FUNCTION_BLOCK Handling_Teach EXTENDS TcoCore.TcoSequencer
VAR
	_o : TcoCore.TcoSequencerObserver(THIS^);	
	_dialog : TcoCore.TcoDialog(THIS^);
END_VAR

PROPERTY Components : REFERENCE TO Handling_Components
GET
VAR
    _parent : POINTER TO Handling;
END_VAR
IF __QUERYPOINTER(_ParentObject,_parent) THEN // Check if _Parent is Station001
	Components REF= _parent^._components;              // If the check is successful dereference a pointer. simlar to THIS^ or SUPER^
END_IF
END_GET
END_PROPERTY

(*~
	<docu>
		<summary>
			Main method of the sequener. Custom code needs to be placed here. The sequencer is executed by call of InstanceName.Run() method.
			This method is abstract, and it must be overridden in derived block.
		</summary>
	</docu>
~*)
METHOD PROTECTED  Main : BOOL
VAR
	test: TcEventEntry;
	answer : TcoCore.eCustomizedDialogAnswer;
	_answer: STRING(INT#3);
END_VAR
THIS^.Observer := _o;

IF (Step(0, TRUE, 'MOVE HORIZONTAL TO LOAD')) THEN
    //--------------------------------------------
	
	_dialog.Show()
			.WithType(eDialogType.Question)				
			.WithCaption('Ready to go?')
			.WithText('Do you really want to start movements? Do we go ahead?')			
			.WithYesNo();
			
	
	IF(_dialog.Answer = TcoCore.eDialogAnswer.Yes) THEN RequestStep(100); _dialog.Restore(); END_IF;
    IF(_dialog.Answer = TcoCore.eDialogAnswer.No) THEN RequestStep(200); _dialog.Restore(); END_IF;
	
    //StepCompleteWhen(_StepElapsedTime > T#5S);
    //--------------------------------------------	
END_IF;


IF (Step(100, TRUE, 'YEEEEEEES')) THEN
    //--------------------------------------------	
    StepCompleteWhen(_StepElapsedTime > T#10S);
    //--------------------------------------------		
END_IF;

IF (Step(200, TRUE, 'NOOOOOOO')) THEN
    //--------------------------------------------	
    StepCompleteWhen(_StepElapsedTime > T#10S);
    //--------------------------------------------		
END_IF;


IF (Step(300, TRUE, 'GROUND MODE COMPLETE')) THEN
    //--------------------------------------------
    //--------------------------------------------	
END_IF;
END_METHOD

END_FUNCTION_BLOCK

(* stored: Version 1.1.0.1
   POU Handling_Teach: Id {c6bc81c9-24ed-4013-a8cd-1c99761ef1ec}, SpecialFunc None
   Property Components: Id {2ff515fa-4b61-48de-ab10-febd461be29a}
   Get Get: Id {938ef0c4-3450-4fb1-81fc-42fdf18de2d7}
   Method Main: Id {de027f2d-ad11-47fa-8dd5-bca0c1f282cc} *)
